INTERFACE ITcoSyncUnit

PROPERTY DataInvalid : BOOL
GET
END_GET
END_PROPERTY

PROPERTY DataValid : BOOL
GET
END_GET
END_PROPERTY

PROPERTY HasSomeIssue : BOOL
GET
END_GET
END_PROPERTY

PROPERTY State : SyncUnitState
GET
END_GET
END_PROPERTY

END_INTERFACE

(* stored: Version 1.1.0.1, ProductVersion 3.1.4024.9
   Itf ITcoSyncUnit: Id {c1b89f76-922c-088d-334c-ef80de38bd6f}
   Property DataInvalid: Id {bbc3ff26-73c9-0418-3842-defd4a48f483}
   Get Get: Id {6f0ddb17-4b82-0639-16ec-779db907ab1e}
   Property DataValid: Id {ae325923-0c82-09dc-32de-eed0138c389b}
   Get Get: Id {f4e5e7ab-dc12-028c-2002-4947562258b6}
   Property HasSomeIssue: Id {dd8ca02c-dd6a-01a2-243d-537f2629f408}
   Get Get: Id {adcd6f78-6310-0e9e-33e9-98cc5e4eb673}
   Property State: Id {572e58cc-87a0-0880-0b2b-92ab534973c4}
   Get Get: Id {b08ac7bf-dabc-0f62-14d7-61c94010bd7a} *)
